///////////
// Structure For Battery Racks. Main Operating Data to be saved ( ex: OPC ) .  
//////////
TYPE CELL :
STRUCT
	
	




END_STRUCT
END_TYPE

(* stored: Version 1.1.0.1, ProductVersion 3.1.4024.6
   DUT CELL: Id {e8bc64e2-20f3-4d06-95cf-ebfd9dc257d8} *)
